PROGRAM POU_ClearAxesErrors
VAR
	fbAxis1Reset:MC_Reset;
	fbAxis2Reset:MC_Reset;
	fbAxis3Reset:MC_Reset;
	fbAxis4Reset:MC_Reset;
	fbAxis5Reset:MC_Reset;
	fbAxis6Reset:MC_Reset;
	END_VAR


fbAxis1Reset(
	Axis:= Axis1, 
	Execute:=bReSetMotor , 
	Done=>bReset1Done , 
	Busy=> , 
	Error=> , 
	ErrorID=> );
	
fbAxis2Reset(
	Axis:= Axis2, 
	Execute:=bReSetMotor , 
	Done=>bReset2Done , 
	Busy=> , 
	Error=> , 
	ErrorID=> );
	
fbAxis3Reset(
	Axis:= Axis3, 
	Execute:=bReSetMotor , 
	Done=>bReset3Done , 
	Busy=> , 
	Error=> , 
	ErrorID=> );
	
fbAxis4Reset(
	Axis:= Axis4, 
	Execute:=bReSetMotor , 
	Done=>bReset4Done , 
	Busy=> , 
	Error=> , 
	ErrorID=> );
	
fbAxis5Reset(
	Axis:= Axis5, 
	Execute:=bReSetMotor , 
	Done=>bReset5Done , 
	Busy=> , 
	Error=> , 
	ErrorID=> );
	
fbAxis6Reset(
	Axis:= Axis6, 
	Execute:=bReSetMotor , 
	Done=>bReset6Done , 
	Busy=> , 
	Error=> , 
	ErrorID=> );

END_PROGRAM

(* stored: Version 1.1.0.1, ProductVersion 3.1.4022.18
   POU POU_ClearAxesErrors: Id {bbcc169f-f8a9-4120-a204-83889109b6fb}, SpecialFunc None *)
